Fanuc KAREL source: kt00044.KL

-- PROVISIONAL review KL for V940-1; original PC SHA256 0dc887a6c5034ad79fb11844b8bb9b56fbef8d205d2c4540dbbb4384b5587eee
-- Incomplete behavior may be omitted. Consult companion uncertainty JSON. Do not deploy.
PROGRAM KT00044
%NOLOCKGROUP
VAR
  R1 : REAL
  R2 : REAL
  OUT : REAL
BEGIN
  -- V9_ZERO_TABLE_METADATA_HINT layout=0001; no indexed target words; source/name/runtime held
  -- UNRESOLVED_PC offsets 5-16; opcodes 2E,23
  -- UNRESOLVED_PC offsets 21-32; opcodes 2E,23
  -- UNRESOLVED_PC offsets 37-48; opcodes 2E,23
  -- UNRESOLVED_PC offsets 53-64; opcodes 2E,23
  -- UNRESOLVED_PC offsets 69-88; opcodes 21,21,6A,23
  -- UNRESOLVED_PC offsets 93-97; opcodes 7F
END KT00044
